{attribute 'hide'}
FUNCTION_BLOCK UCS
VAR_INPUT
	oid														:	UDINT := 0;		//Object identifier
	vTranslation 											:	VECTOR;
 	vRotation 												:	VECTOR;
	Valid													:	BOOL := FALSE;
END_VAR
VAR_OUTPUT
END_VAR
VAR
END_VAR

METHOD delete : BOOL
VAR_INPUT
END_VAR
MEMSET(ADR(vTranslation),0,SIZEOF(vTranslation));
MEMSET(ADR(VRotation),0,SIZEOF(VRotation));
oid 													:= 0;
delete	:= TRUE;
END_METHOD

END_FUNCTION_BLOCK

(* stored: Version 1.1.0.1, ProductVersion 3.1.4024.6
   POU UCS: Id {6f0af4b2-3151-4bea-8a8f-c47090bfc4a2}, SpecialFunc None
   Method delete: Id {d382f36b-ea83-408c-8666-d9fb9aa0877f} *)
